PROGRAM TEST
VAR
END_VAR

GVL.ENCODER_1_RAW_COUNTS;

END_PROGRAM

(* stored: Version 1.1.0.1, ProductVersion 3.1.4024.12
   POU TEST: Id {9e6940e2-7b3f-425d-b76c-928c06cc9bd2}, SpecialFunc None *)
